(* Logix 5000 project; controller Commerford_topping_5477_V3 vendor 1 type 14 code 222 rev 33.11; software revision 33.02; part 5 of 6 *)
(* tags used below, declared in another part *)
   HMI_SAF_Reset : BOOL;   // Safety reset for HMI
(* UN6_EM4_Color_3, continued *)

ROUTINE Main   (* ladder *)
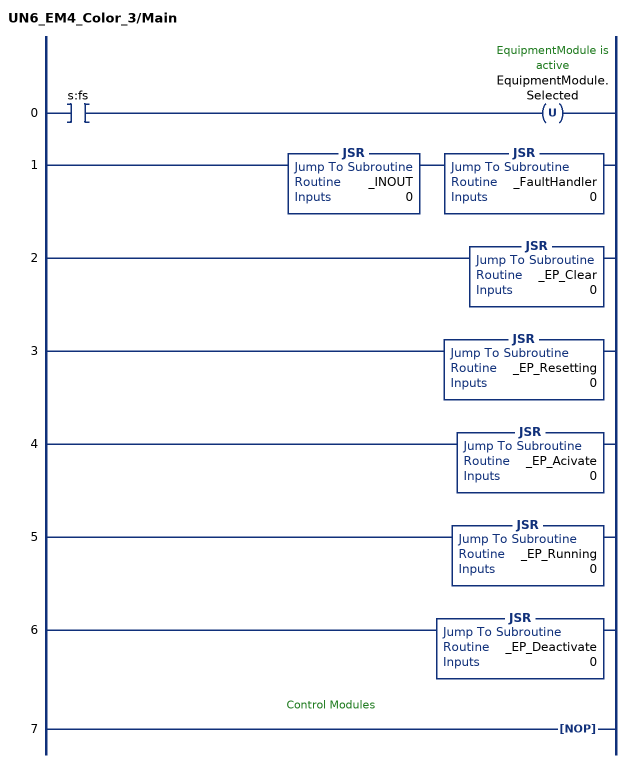
   0: XIC(s:fs)OTU(EquipmentModule.Selected);
   1: JSR(_INOUT,0)JSR(_FaultHandler,0);
   2: JSR(_EP_Clear,0);
   3: JSR(_EP_Resetting,0);
   4: JSR(_EP_Acivate,0);
   5: JSR(_EP_Running,0);
   6: JSR(_EP_Deactivate,0);
   // Control Modules
   7: NOP();
END_ROUTINE
END_PROGRAM

PROGRAM UN6_EM5_No_Color   (* main routine Main *)
// No_Color, generated by G.E.M
VAR
   _Cmd_Activate : BOOL;
   _Cmd_ClearFaults : BOOL;
   _Cmd_Deactivate : BOOL;
   _Cmd_Reset : BOOL;
   _Sts_AcivateSeq_PC : BOOL;
   _Sts_ClearSeq_PC : BOOL;
   _Sts_DeactivateSeq_PC : BOOL;
   _Sts_Execute_PC : BOOL;
   _Sts_ResetSeq_PC : BOOL;
END_VAR
VAR {public}
   EquipmentModule : EquipmentModule := (Selected := 1, State_in := 2#0000_0000_0000_0000_0000_0000_0000_0101, State_out := 2#0000_0000_0000_0000_0000_0000_0000_0001, _SEQ.Clearing := -1, _SEQ.Activating := -1, _SEQ.Deactivating := -1, _SEQ.Resetting := -1);
        .State_in.1   // Clearing
END_VAR

ROUTINE _EP_Acivate   (* ladder *)
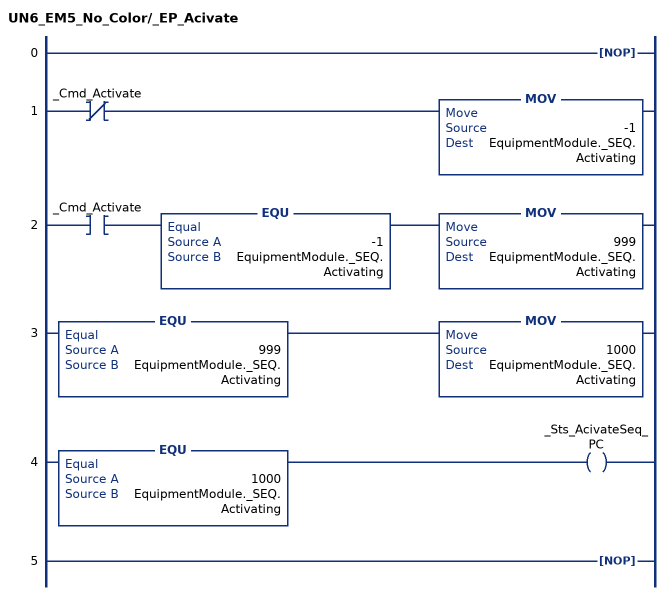
   0: NOP();
   1: XIO(_Cmd_Activate)MOV(-1,EquipmentModule._SEQ.Activating);
   2: XIC(_Cmd_Activate)EQU(-1,EquipmentModule._SEQ.Activating)MOV(999,EquipmentModule._SEQ.Activating);
   3: EQU(999,EquipmentModule._SEQ.Activating)MOV(1000,EquipmentModule._SEQ.Activating);
   4: EQU(1000,EquipmentModule._SEQ.Activating)OTE(_Sts_AcivateSeq_PC);
   5: NOP();
END_ROUTINE

ROUTINE _EP_Clear   (* ladder *)
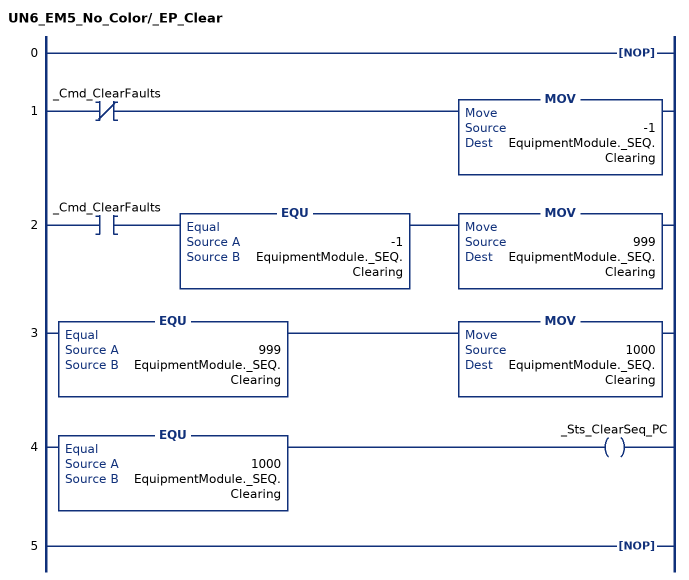
   0: NOP();
   1: XIO(_Cmd_ClearFaults)MOV(-1,EquipmentModule._SEQ.Clearing);
   2: XIC(_Cmd_ClearFaults)EQU(-1,EquipmentModule._SEQ.Clearing)MOV(999,EquipmentModule._SEQ.Clearing);
   3: EQU(999,EquipmentModule._SEQ.Clearing)MOV(1000,EquipmentModule._SEQ.Clearing);
   4: EQU(1000,EquipmentModule._SEQ.Clearing)OTE(_Sts_ClearSeq_PC);
   5: NOP();
END_ROUTINE

ROUTINE _EP_Deactivate   (* ladder *)
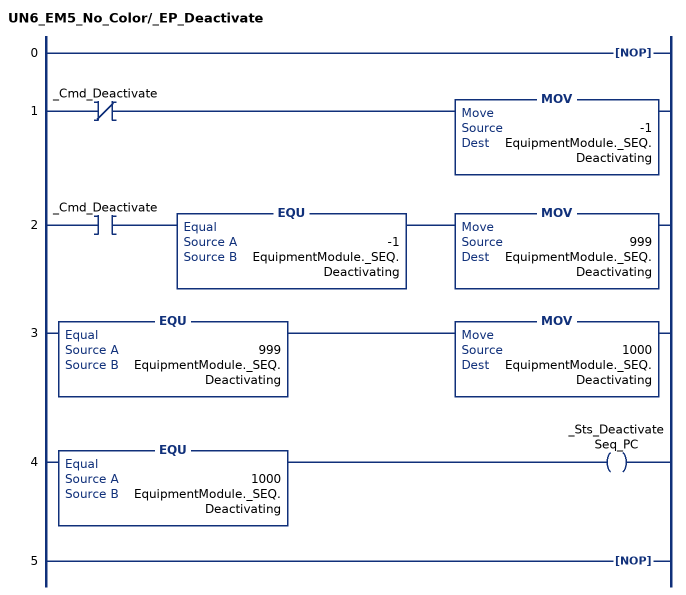
   0: NOP();
   1: XIO(_Cmd_Deactivate)MOV(-1,EquipmentModule._SEQ.Deactivating);
   2: XIC(_Cmd_Deactivate)EQU(-1,EquipmentModule._SEQ.Deactivating)MOV(999,EquipmentModule._SEQ.Deactivating);
   3: EQU(999,EquipmentModule._SEQ.Deactivating)MOV(1000,EquipmentModule._SEQ.Deactivating);
   4: EQU(1000,EquipmentModule._SEQ.Deactivating)OTE(_Sts_DeactivateSeq_PC);
   5: NOP();
END_ROUTINE

ROUTINE _EP_Resetting   (* ladder *)
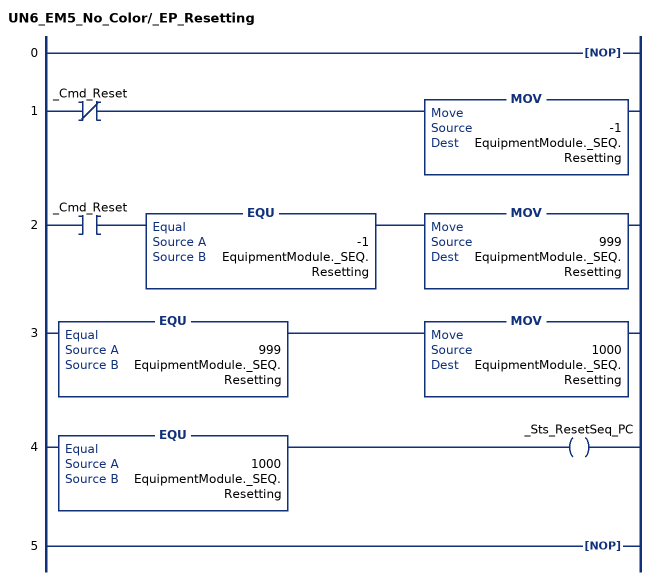
   0: NOP();
   1: XIO(_Cmd_Reset)MOV(-1,EquipmentModule._SEQ.Resetting);
   2: XIC(_Cmd_Reset)EQU(-1,EquipmentModule._SEQ.Resetting)MOV(999,EquipmentModule._SEQ.Resetting);
   3: EQU(999,EquipmentModule._SEQ.Resetting)MOV(1000,EquipmentModule._SEQ.Resetting);
   4: EQU(1000,EquipmentModule._SEQ.Resetting)OTE(_Sts_ResetSeq_PC);
   5: NOP();
END_ROUTINE

ROUTINE _EP_Running   (* ladder *)
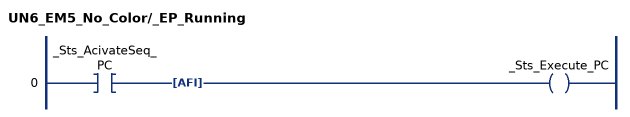
   0: XIC(_Sts_AcivateSeq_PC)AFI()OTE(_Sts_Execute_PC);
END_ROUTINE

ROUTINE _FaultHandler   (* ladder *)
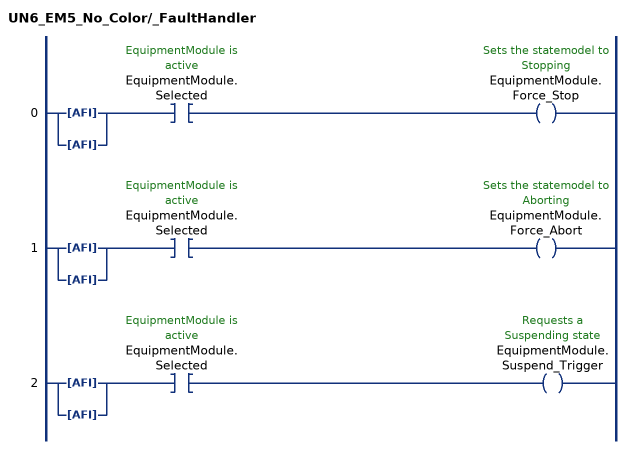
   0: [AFI() ,AFI() ]XIC(EquipmentModule.Selected)OTE(EquipmentModule.Force_Stop);
   1: [AFI() ,AFI() ]XIC(EquipmentModule.Selected)OTE(EquipmentModule.Force_Abort);
   2: [AFI() ,AFI() ]XIC(EquipmentModule.Selected)OTE(EquipmentModule.Suspend_Trigger);
END_ROUTINE

ROUTINE _INOUT   (* ladder *)
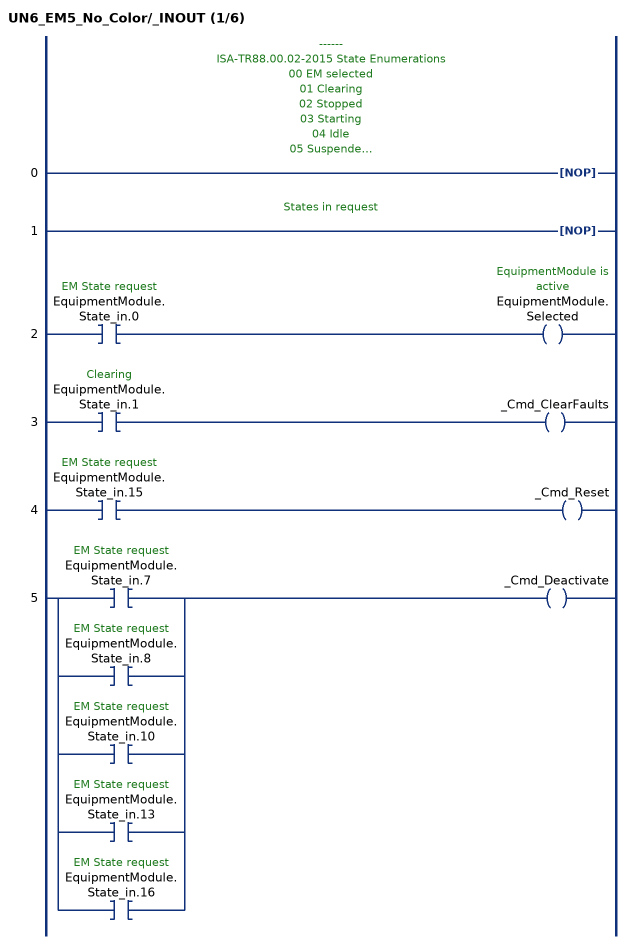
   // ------
   // ISA-TR88.00.02-2015 State Enumerations
   // 00 EM selected
   // 01 Clearing
   // 02 Stopped
   // 03 Starting
   // 04 Idle
   // 05 Suspended
   // 06 Execute
   // 07 Stopping
   // 08 Aborting
   // 09 Aborted
   // 10 Holding
   // 11 Held
   // 12 UnHolding
   // 13 Suspending
   // 14 Unsuspending
   // 15 Resetting
   // 16 Completing
   // 17 Complete
   // 18 Undefined
   // 19 Undefined
   // 20 Suspend trigger
   // 21 Faulted
   // 22 Force stop
   // 23 Force abort
   // 24 Reset signal
   // 31 Undefined
   // ------
   0: NOP();
   // States in request
   1: NOP();
   2: XIC(EquipmentModule.State_in.0)OTE(EquipmentModule.Selected);
   3: XIC(EquipmentModule.State_in.1)OTE(_Cmd_ClearFaults);
   4: XIC(EquipmentModule.State_in.15)OTE(_Cmd_Reset);
   5: [XIC(EquipmentModule.State_in.7) ,XIC(EquipmentModule.State_in.8) ,XIC(EquipmentModule.State_in.10) ,XIC(EquipmentModule.State_in.13) ,XIC(EquipmentModule.State_in.16) ]OTE(_Cmd_Deactivate);
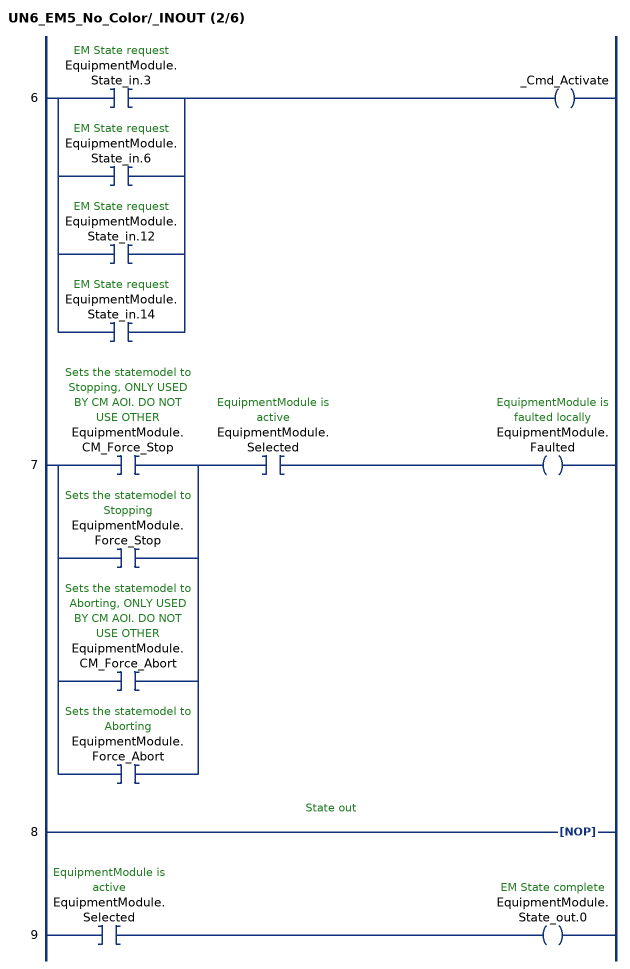
   6: [XIC(EquipmentModule.State_in.3) ,XIC(EquipmentModule.State_in.6) ,XIC(EquipmentModule.State_in.12) ,XIC(EquipmentModule.State_in.14) ]OTE(_Cmd_Activate);
   7: [XIC(EquipmentModule.CM_Force_Stop) ,XIC(EquipmentModule.Force_Stop) ,XIC(EquipmentModule.CM_Force_Abort) ,XIC(EquipmentModule.Force_Abort) ]XIC(EquipmentModule.Selected)OTE(EquipmentModule.Faulted);
   // State out
   8: NOP();
   9: XIC(EquipmentModule.Selected)OTE(EquipmentModule.State_out.0);
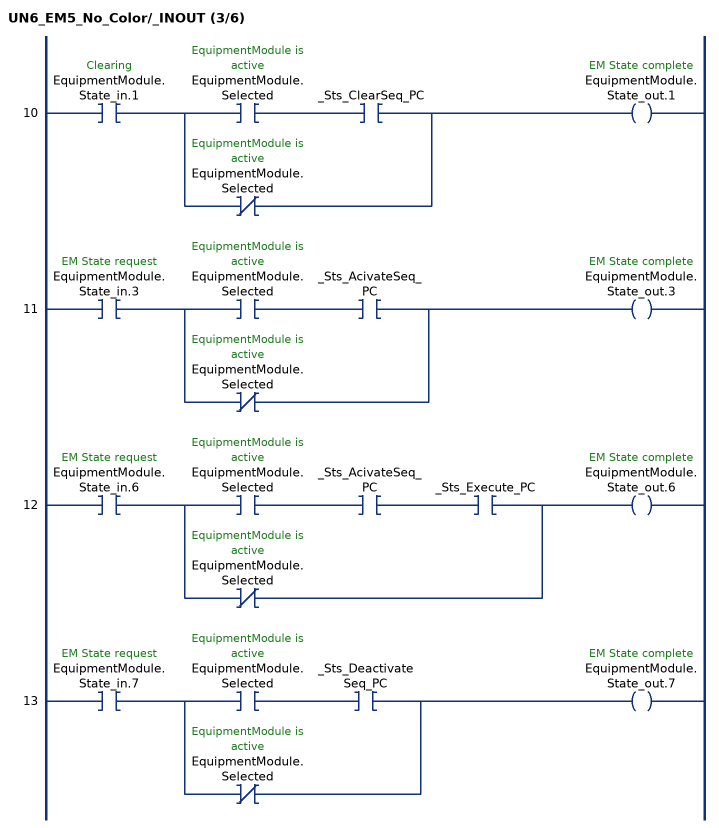
   10: XIC(EquipmentModule.State_in.1)[XIC(EquipmentModule.Selected) XIC(_Sts_ClearSeq_PC) ,XIO(EquipmentModule.Selected) ]OTE(EquipmentModule.State_out.1);
   11: XIC(EquipmentModule.State_in.3)[XIC(EquipmentModule.Selected) XIC(_Sts_AcivateSeq_PC) ,XIO(EquipmentModule.Selected) ]OTE(EquipmentModule.State_out.3);
   12: XIC(EquipmentModule.State_in.6)[XIC(EquipmentModule.Selected) XIC(_Sts_AcivateSeq_PC) XIC(_Sts_Execute_PC) ,XIO(EquipmentModule.Selected) ]OTE(EquipmentModule.State_out.6);
   13: XIC(EquipmentModule.State_in.7)[XIC(EquipmentModule.Selected) XIC(_Sts_DeactivateSeq_PC) ,XIO(EquipmentModule.Selected) ]OTE(EquipmentModule.State_out.7);
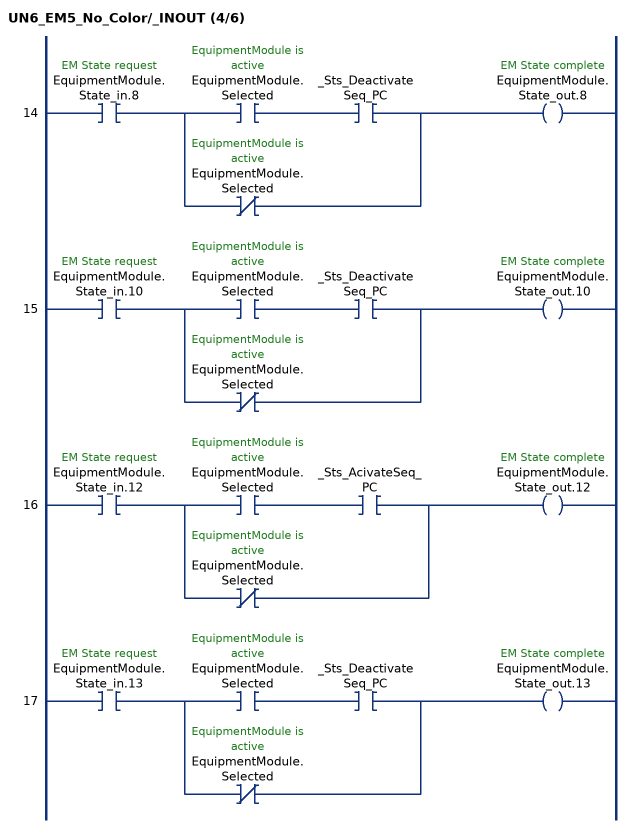
   14: XIC(EquipmentModule.State_in.8)[XIC(EquipmentModule.Selected) XIC(_Sts_DeactivateSeq_PC) ,XIO(EquipmentModule.Selected) ]OTE(EquipmentModule.State_out.8);
   15: XIC(EquipmentModule.State_in.10)[XIC(EquipmentModule.Selected) XIC(_Sts_DeactivateSeq_PC) ,XIO(EquipmentModule.Selected) ]OTE(EquipmentModule.State_out.10);
   16: XIC(EquipmentModule.State_in.12)[XIC(EquipmentModule.Selected) XIC(_Sts_AcivateSeq_PC) ,XIO(EquipmentModule.Selected) ]OTE(EquipmentModule.State_out.12);
   17: XIC(EquipmentModule.State_in.13)[XIC(EquipmentModule.Selected) XIC(_Sts_DeactivateSeq_PC) ,XIO(EquipmentModule.Selected) ]OTE(EquipmentModule.State_out.13);
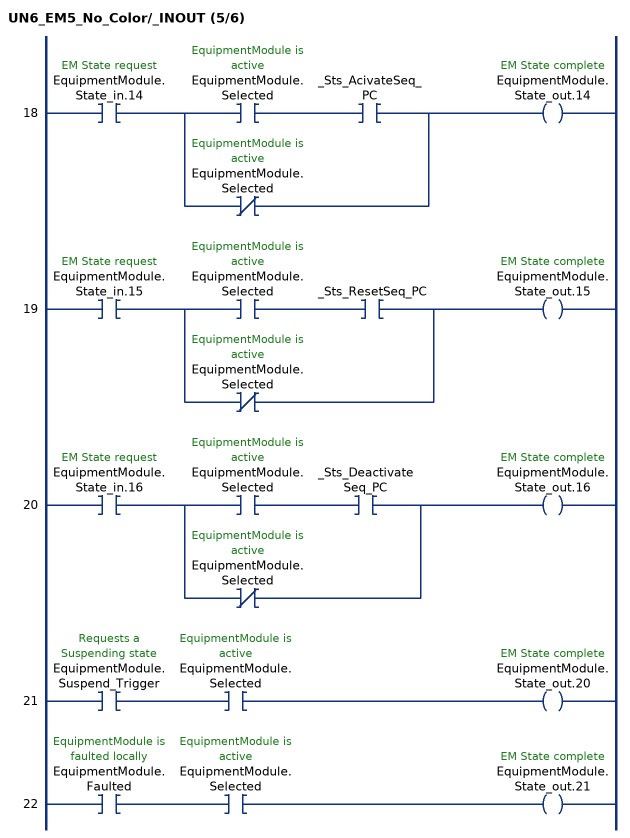
   18: XIC(EquipmentModule.State_in.14)[XIC(EquipmentModule.Selected) XIC(_Sts_AcivateSeq_PC) ,XIO(EquipmentModule.Selected) ]OTE(EquipmentModule.State_out.14);
   19: XIC(EquipmentModule.State_in.15)[XIC(EquipmentModule.Selected) XIC(_Sts_ResetSeq_PC) ,XIO(EquipmentModule.Selected) ]OTE(EquipmentModule.State_out.15);
   20: XIC(EquipmentModule.State_in.16)[XIC(EquipmentModule.Selected) XIC(_Sts_DeactivateSeq_PC) ,XIO(EquipmentModule.Selected) ]OTE(EquipmentModule.State_out.16);
   21: XIC(EquipmentModule.Suspend_Trigger)XIC(EquipmentModule.Selected)OTE(EquipmentModule.State_out.20);
   22: XIC(EquipmentModule.Faulted)XIC(EquipmentModule.Selected)OTE(EquipmentModule.State_out.21);
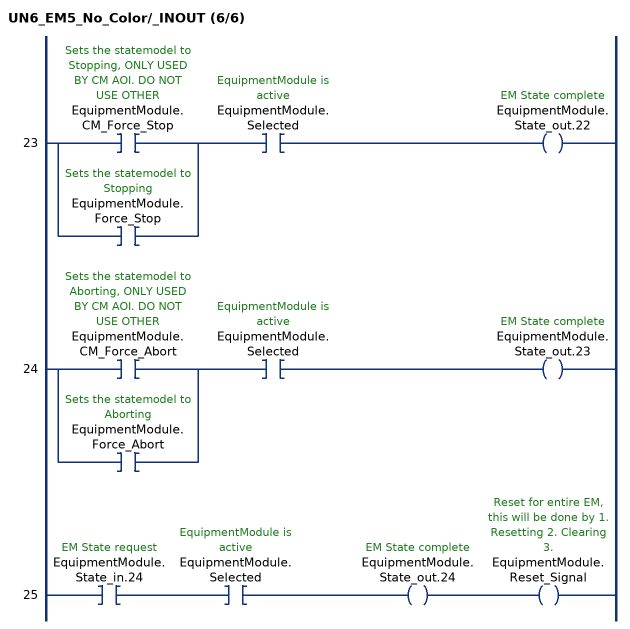
   23: [XIC(EquipmentModule.CM_Force_Stop) ,XIC(EquipmentModule.Force_Stop) ]XIC(EquipmentModule.Selected)OTE(EquipmentModule.State_out.22);
   24: [XIC(EquipmentModule.CM_Force_Abort) ,XIC(EquipmentModule.Force_Abort) ]XIC(EquipmentModule.Selected)OTE(EquipmentModule.State_out.23);
   25: XIC(EquipmentModule.State_in.24)XIC(EquipmentModule.Selected)OTE(EquipmentModule.State_out.24)OTE(EquipmentModule.Reset_Signal);
END_ROUTINE

ROUTINE Main   (* ladder *)
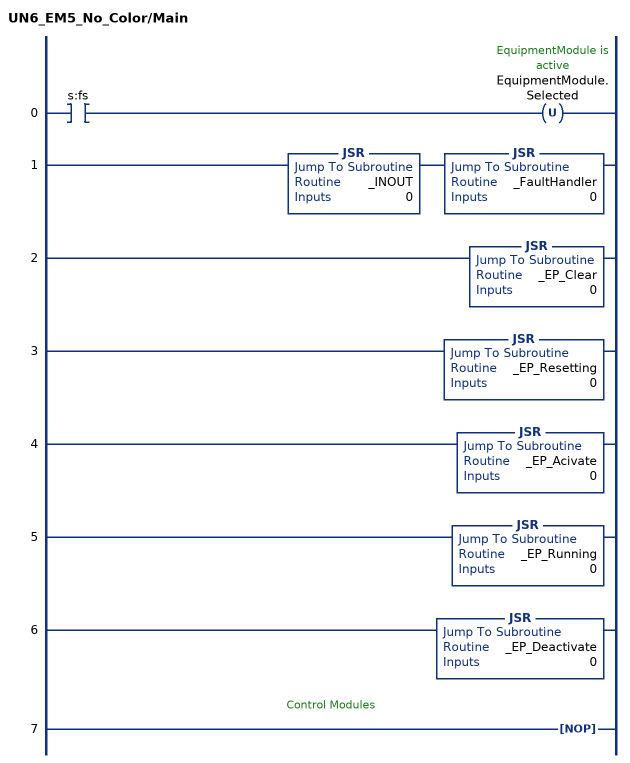
   0: XIC(s:fs)OTU(EquipmentModule.Selected);
   1: JSR(_INOUT,0)JSR(_FaultHandler,0);
   2: JSR(_EP_Clear,0);
   3: JSR(_EP_Resetting,0);
   4: JSR(_EP_Acivate,0);
   5: JSR(_EP_Running,0);
   6: JSR(_EP_Deactivate,0);
   // Control Modules
   7: NOP();
END_ROUTINE
END_PROGRAM

PROGRAM UN6_Object   (* main routine PackML *)
VAR
   Debug : DINT;
   EMStates : DINT[32] := ([1] := 1, [2] := 1, [3] := 1);
   HMI_Show_Tags : BOOL;   // Show HMI tags
   MachineStates : Packml_States := (Aborting := 1, Aborted := 1, Clearing := 1, Stopping := 1, Stopped := 1, Resetting := 1, Idle := 1, Starting := 1, Execute := 1, Holding := 1, Held := 1, Unholding := 1, Suspending := 1, Suspended := 1, Unsuspending := 1, Completing := 1, Complete := 1);   // Active machine states
   OEM_AutomaticUnsuspend : BOOL := 1;
   Packml_RequestClear : ISA_TR_88_00_02_StateChangeRequest := (RequestCmd := 9);
   Packml_RequestState : ISA_TR_88_00_02_StateChangeRequest := (RequestCmd := 7);
   Packml_RequestUnsuspend : ISA_TR_88_00_02_StateChangeRequest := (RequestCmd := 7);
   Proces : ProcessHandler := (Process_ID := 1);
END_VAR
VAR {public}
   EM : EquipmentModule_Link[6];
   Master_Recipe : MasterRecipeSelect := (Recipe := '286379852(1),287794021(2),288750792(3),', SelectedRecipeNum := 1, SelectedProces := 2, Process := 'Production(1),Pre-Production(2),');
   PackML : ISA_TR_88_00_02 := (Sts_SC_Status := 2#1111_1111_1111_1111_1111_1111_1111_0001, Sts_Aborted := 1, Sts_Automatic := 1, Process_Selected := 2, Sts_MachineFaulted := 1);
   PML_Machine : PACKMLv30 := (Command.CntrlCmd := 7, Status.UnitModeCurrent := 1, Status.StateCurrent := 9, Status.StateRequested := 9, Status.MachSpeed := 1.0, Status.UnitFaulted := 1, Admin.ModeCurrentTime[1] := 79332, Admin.ModeCumulativeTime[1] := 212, Admin.StateCurrentTime[1].Mode[9] := 212, Admin.StateCumulativeTime[1].Mode[1] := 570, Admin.StateCumulativeTime[1].Mode[2] := 74675, Admin.StateCumulativeTime[1].Mode[3] := 101, Admin.StateCumulativeTime[1].Mode[4] := 16868, Admin.StateCumulativeTime[1].Mode[5] := 146, Admin.StateCumulativeTime[1].Mode[6] := 78246, Admin.StateCumulativeTime[1].Mode[7] := 950, Admin.StateCumulativeTime[1].Mode[8] := 307, Admin.StateCumulativeTime[1].Mode[9] := 252889, Admin.StateCumulativeTime[1].Mode[10] := 25, Admin.StateCumulativeTime[1].Mode[11] := 22006, Admin.StateCumulativeTime[1].Mode[12] := 7, Admin.StateCumulativeTime[1].Mode[13] := 54, Admin.StateCumulativeTime[1].Mode[14] := 58, Admin.StateCumulativeTime[1].Mode[15] := 1580, Admin.StateCumulativeTime[1].Mode[16] := 23, Admin.StateCumulativeTime[1].Mode[17] := 238, Admin.StateCumulativeTime[2].Mode[2] := 96, Admin.StateCumulativeTime[2].Mode[4] := 147, Admin.StateCumulativeTime[2].Mode[9] := 10, Admin.StateCumulativeTime[2].Mode[15] := 1, Admin.StateCumulativeTime[3].Mode[1] := 2, Admin.StateCumulativeTime[3].Mode[2] := 121062, Admin.StateCumulativeTime[3].Mode[4] := 247936, Admin.StateCumulativeTime[3].Mode[6] := 12, Admin.StateCumulativeTime[3].Mode[9] := 3256, Admin.StateCumulativeTime[3].Mode[15] := 6, Admin.AccTimeSinceReset := 791, Admin.PACDateTime.Date := 1699868570913630, Admin.PACDateTime.Time := 1699868570913630);   // Packtag machine info
   ProcessStates : DINT[32] := ([2] := 1);
   Recipe : RecipeManager[4] := ([0].i := 2, [0].RecipeSize := 15, [0].RecipeSettingsSize := 20, [1].i := 10, [1].RecipeSize := 20, [1].RecipeSettingsSize := 100, [1].SelectedRecipeNum := 1, [1].Str_Temp := '-1971450705(1),', [1].wrk_UploadTempValue_LINT := 899256806149295, [1].wrk_UploadTempValue_DINT := -1971450705, [1].j := 11, [1].Wrk_TempNum := 1, [1].wrk_TempString := '19', [1].d_Update_CurrentlyRunningRecipe := 1, [2].i := 10, [2].RecipeSize := 20, [2].RecipeSettingsSize := 100, [2].SelectedRecipeNum := 1, [2].RecipeList := '286379852(1),287794021(2),288750792(3),', [2].wrk_RecipeList[1].Name := '286379852', [2].wrk_RecipeList[1].TimeSaved := 896321306349388, [2].wrk_RecipeList[2].Name := '287794021', [2].wrk_RecipeList[2].TimeSaved := 896321307763557, [2].wrk_RecipeList[3].Name := '288750792', [2].wrk_RecipeList[3].TimeSaved := 896321308720328, [2].Str_SelectedRecipe := '286379852', [2].Str_Temp := '288750792(3),', [2].wrk_UploadTempValue_LINT := 896321315117083, [2].wrk_UploadTempValue_DINT := 295147547, [2].j := 100, [2].Str_CurrentlyRunningRecipe := '286379852', [2].Wrk_TempNum := 27, [2].wrk_TempString := '19', [2].HMI_Config_Rename_Input := '286379852', [2].Time_SelectedRecipe := 896321306349388, [2].d_Update_CurrentlyRunningRecipe := 1);
END_VAR

ROUTINE EquipmentModule_Management   (* ladder *)
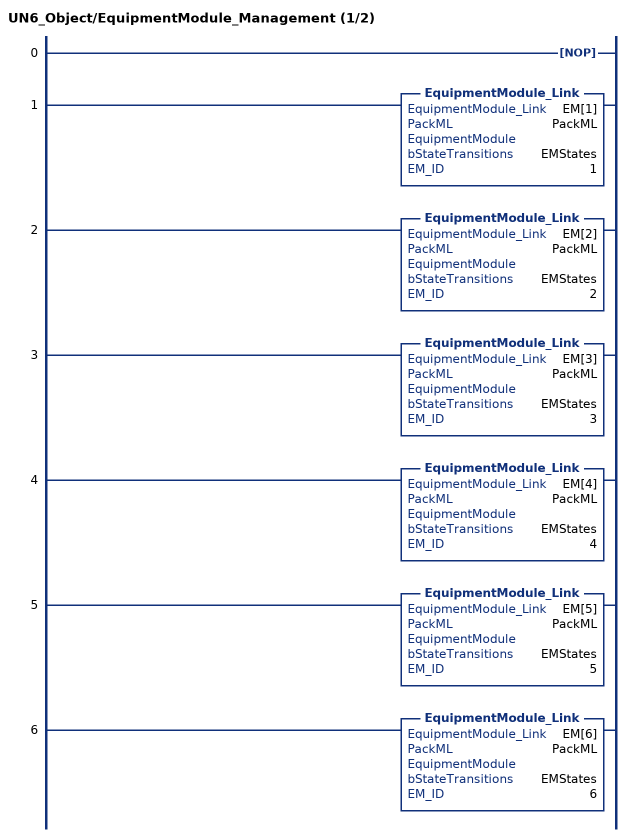
   0: NOP();
   1: EquipmentModule_Link(EM[1],PackML,,EMStates,1);
   2: EquipmentModule_Link(EM[2],PackML,,EMStates,2);
   3: EquipmentModule_Link(EM[3],PackML,,EMStates,3);
   4: EquipmentModule_Link(EM[4],PackML,,EMStates,4);
   5: EquipmentModule_Link(EM[5],PackML,,EMStates,5);
   6: EquipmentModule_Link(EM[6],PackML,,EMStates,6);
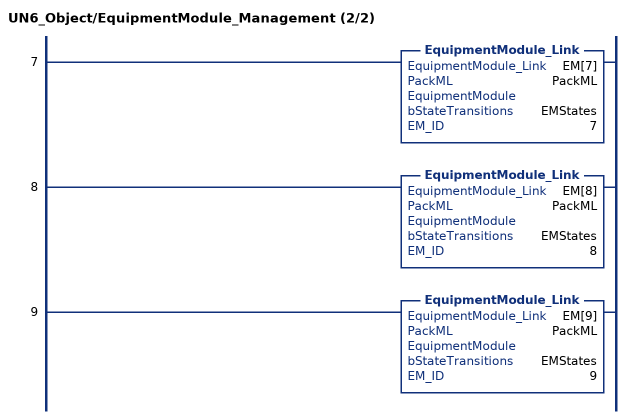
   7: EquipmentModule_Link(EM[7],PackML,,EMStates,7);
   8: EquipmentModule_Link(EM[8],PackML,,EMStates,8);
   9: EquipmentModule_Link(EM[9],PackML,,EMStates,9);
END_ROUTINE

ROUTINE PackML   (* ladder *)
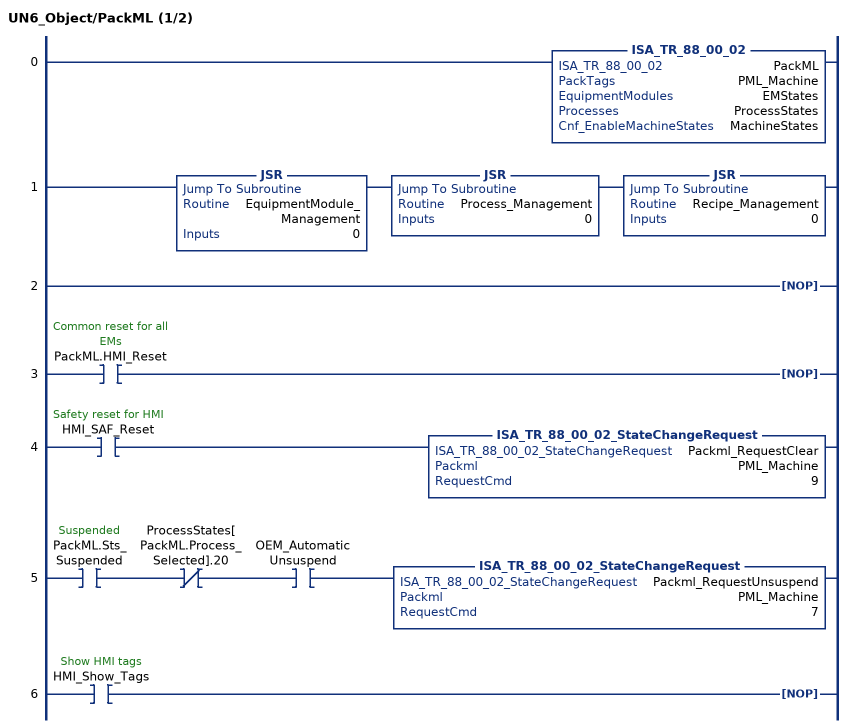
   0: ISA_TR_88_00_02(PackML,PML_Machine,EMStates,ProcessStates,MachineStates);
   1: JSR(EquipmentModule_Management,0)JSR(Process_Management,0)JSR(Recipe_Management,0);
   2: NOP();
   3: XIC(PackML.HMI_Reset)NOP();
   4: XIC(HMI_SAF_Reset)ISA_TR_88_00_02_StateChangeRequest(Packml_RequestClear,PML_Machine,9);
   5: XIC(PackML.Sts_Suspended)XIO(ProcessStates[PackML.Process_Selected].20)XIC(OEM_AutomaticUnsuspend)ISA_TR_88_00_02_StateChangeRequest(Packml_RequestUnsuspend,PML_Machine,7);
   6: XIC(HMI_Show_Tags)NOP();
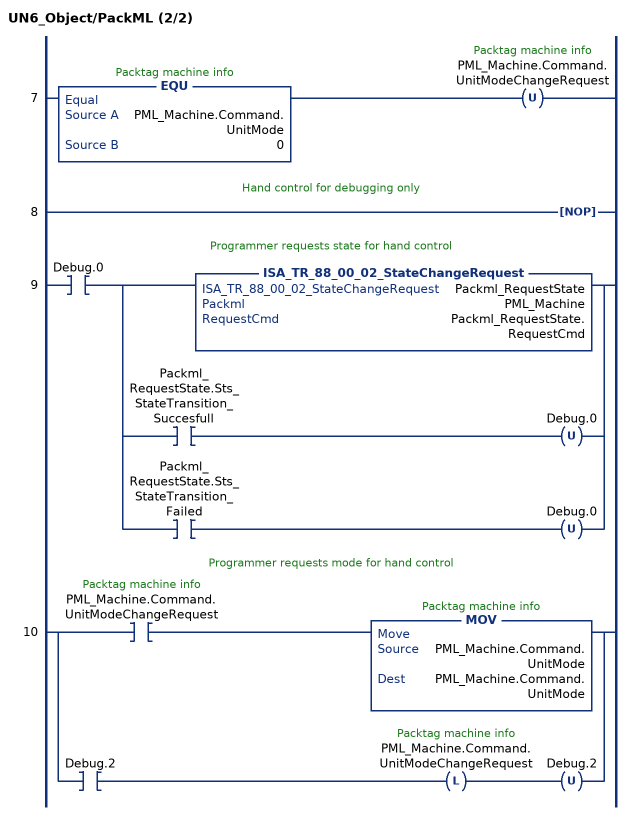
   7: EQU(PML_Machine.Command.UnitMode,0)OTU(PML_Machine.Command.UnitModeChangeRequest);
   // Hand control for debugging only
   8: NOP();
   // Programmer requests state for hand control
   9: XIC(Debug.0)[ISA_TR_88_00_02_StateChangeRequest(Packml_RequestState,PML_Machine,Packml_RequestState.RequestCmd) ,XIC(Packml_RequestState.Sts_StateTransition_Succesfull) OTU(Debug.0) ,XIC(Packml_RequestState.Sts_StateTransition_Failed) OTU(Debug.0) ];
   // Programmer requests mode for hand control
   10: [XIC(PML_Machine.Command.UnitModeChangeRequest) MOV(PML_Machine.Command.UnitMode,PML_Machine.Command.UnitMode) ,XIC(Debug.2) OTL(PML_Machine.Command.UnitModeChangeRequest) OTU(Debug.2) ];
END_ROUTINE
